// Tankregelung SCL - generated by build-scl.ps1
// Do not edit directly; modify src/tank/*.scl and rebuild.

// --- types\tank_mode.scl ---
TYPE "TankMode" :
(
    Off := 0,
    Manual := 1,
    Auto := 2
);
END_TYPE

// --- data_blocks\db_hmi_tank.scl ---
DATA_BLOCK "DB_HMI_Tank"
{ S7_Optimized_Access := 'TRUE' }
VERSION : 0.1
VAR
    // HMI commands
    Mode : Int := 0;
    StartAuto : Bool := FALSE;
    Stop : Bool := FALSE;
    ManualFill : Bool := FALSE;
    ManualDrain : Bool := FALSE;
    ResetFault : Bool := FALSE;

    // HMI parameters
    SetpointPct : Real := 60.0;
    HysteresisPct : Real := 3.0;
    LowLowPct : Real := 5.0;
    HighHighPct : Real := 95.0;

    // PLC/HMI status
    LevelPct : Real := 20.0;
    FillValveCmd : Bool := FALSE;
    DrainValveCmd : Bool := FALSE;
    AutoActive : Bool := FALSE;
    Fault : Bool := FALSE;
    AlarmLowLow : Bool := FALSE;
    AlarmHighHigh : Bool := FALSE;
    StatusText : String[80] := 'Aus';
END_VAR
BEGIN
END_DATA_BLOCK

// --- scl\fb_tank_control.scl ---
FUNCTION_BLOCK "FB_TankControl"
{ S7_Optimized_Access := 'TRUE' }
VERSION : 0.1
VAR_INPUT
    LevelPct : Real;
    Mode : Int;
    StartAuto : Bool;
    Stop : Bool;
    ManualFill : Bool;
    ManualDrain : Bool;
    ResetFault : Bool;
    SetpointPct : Real;
    HysteresisPct : Real;
    LowLowPct : Real;
    HighHighPct : Real;
END_VAR
VAR_OUTPUT
    FillValveCmd : Bool;
    DrainValveCmd : Bool;
    AutoActive : Bool;
    Fault : Bool;
    AlarmLowLow : Bool;
    AlarmHighHigh : Bool;
    StatusText : String[80];
END_VAR
VAR
    FillLatch : Bool;
    SetpointLimited : Real;
    HysteresisLimited : Real;
END_VAR
BEGIN
    // Plausible Bedienwerte begrenzen.
    SetpointLimited := LIMIT(MN := 1.0, IN := SetpointPct, MX := 99.0);
    HysteresisLimited := LIMIT(MN := 0.5, IN := HysteresisPct, MX := 20.0);

    AlarmLowLow := LevelPct <= LowLowPct;
    AlarmHighHigh := LevelPct >= HighHighPct;

    IF AlarmHighHigh THEN
        Fault := TRUE;
    END_IF;

    IF ResetFault AND NOT AlarmHighHigh THEN
        Fault := FALSE;
    END_IF;

    IF Stop OR Fault OR (Mode = 0) THEN
        AutoActive := FALSE;
        FillLatch := FALSE;
    ELSIF (Mode = 2) AND StartAuto THEN
        AutoActive := TRUE;
    END_IF;

    FillValveCmd := FALSE;
    DrainValveCmd := FALSE;

    CASE Mode OF
        0:
            StatusText := 'Aus';

        1:
            AutoActive := FALSE;
            FillLatch := FALSE;
            FillValveCmd := ManualFill AND NOT Fault AND NOT AlarmHighHigh;
            DrainValveCmd := ManualDrain AND NOT ManualFill;

            IF Fault THEN
                StatusText := 'Stoerung';
            ELSE
                StatusText := 'Handbetrieb';
            END_IF;

        2:
            IF AutoActive AND NOT Fault THEN
                IF LevelPct <= (SetpointLimited - HysteresisLimited) THEN
                    FillLatch := TRUE;
                ELSIF LevelPct >= (SetpointLimited + HysteresisLimited) THEN
                    FillLatch := FALSE;
                END_IF;

                FillValveCmd := FillLatch AND NOT AlarmHighHigh;
                DrainValveCmd := FALSE;
                StatusText := 'Automatik aktiv';
            ELSIF Fault THEN
                StatusText := 'Stoerung';
            ELSE
                StatusText := 'Automatik bereit';
            END_IF;

        ELSE
            AutoActive := FALSE;
            FillLatch := FALSE;
            StatusText := 'Ungueltige Betriebsart';
    END_CASE;
END_FUNCTION_BLOCK

// --- scl\fb_tank_sim.scl ---
FUNCTION_BLOCK "FB_TankSim"
{ S7_Optimized_Access := 'TRUE' }
VERSION : 0.1
VAR_INPUT
    Enable : Bool;
    FillValveCmd : Bool;
    DrainValveCmd : Bool;
END_VAR
VAR_IN_OUT
    LevelPct : Real;
END_VAR
VAR
    FillRatePctPerCycle : Real := 0.08;
    DrainRatePctPerCycle : Real := 0.05;
    NaturalOutflowPctPerCycle : Real := 0.01;
END_VAR
BEGIN
    IF Enable THEN
        IF FillValveCmd THEN
            LevelPct := LevelPct + FillRatePctPerCycle;
        END_IF;

        IF DrainValveCmd THEN
            LevelPct := LevelPct - DrainRatePctPerCycle;
        END_IF;

        LevelPct := LevelPct - NaturalOutflowPctPerCycle;
        LevelPct := LIMIT(MN := 0.0, IN := LevelPct, MX := 100.0);
    END_IF;
END_FUNCTION_BLOCK

// --- data_blocks\instance_dbs.scl ---
DATA_BLOCK "FB_TankControl_DB" "FB_TankControl"
{ S7_Optimized_Access := 'TRUE' }
VERSION : 0.1
BEGIN
END_DATA_BLOCK

DATA_BLOCK "FB_TankSim_DB" "FB_TankSim"
{ S7_Optimized_Access := 'TRUE' }
VERSION : 0.1
BEGIN
END_DATA_BLOCK

// --- plc\main.scl ---
ORGANIZATION_BLOCK "Main"
{ S7_Optimized_Access := 'TRUE' }
VERSION : 0.1
VAR_TEMP
END_VAR
BEGIN
    "FB_TankControl_DB"(
        LevelPct := "DB_HMI_Tank".LevelPct,
        Mode := "DB_HMI_Tank".Mode,
        StartAuto := "DB_HMI_Tank".StartAuto,
        Stop := "DB_HMI_Tank".Stop,
        ManualFill := "DB_HMI_Tank".ManualFill,
        ManualDrain := "DB_HMI_Tank".ManualDrain,
        ResetFault := "DB_HMI_Tank".ResetFault,
        SetpointPct := "DB_HMI_Tank".SetpointPct,
        HysteresisPct := "DB_HMI_Tank".HysteresisPct,
        LowLowPct := "DB_HMI_Tank".LowLowPct,
        HighHighPct := "DB_HMI_Tank".HighHighPct,
        FillValveCmd => "DB_HMI_Tank".FillValveCmd,
        DrainValveCmd => "DB_HMI_Tank".DrainValveCmd,
        AutoActive => "DB_HMI_Tank".AutoActive,
        Fault => "DB_HMI_Tank".Fault,
        AlarmLowLow => "DB_HMI_Tank".AlarmLowLow,
        AlarmHighHigh => "DB_HMI_Tank".AlarmHighHigh,
        StatusText => "DB_HMI_Tank".StatusText);

    "FB_TankSim_DB"(
        Enable := TRUE,
        FillValveCmd := "DB_HMI_Tank".FillValveCmd,
        DrainValveCmd := "DB_HMI_Tank".DrainValveCmd,
        LevelPct := "DB_HMI_Tank".LevelPct);
END_ORGANIZATION_BLOCK

